TYPE EL6021_COM_Outputs :
STRUCT
	{attribute addProperty Name "Control"}
	Control AT %Q* : EL6021_Control;
	{attribute addProperty Name "Data"}
	Data  AT %Q* : ARRAY[0..21] OF USINT;
END_STRUCT
END_TYPE

(* stored: Version 1.1.0.1, ProductVersion 3.1.4024.9
   DUT EL6021_COM_Outputs: Id {072a9996-e9b2-0c30-381e-777dcd30b225} *)
